INTERFACE ICylinder EXTENDS __System.IQueryInterface

PROPERTY AtHome : bool
GET
END_GET
END_PROPERTY

PROPERTY AtWork : bool
GET
END_GET
END_PROPERTY

METHOD MoveToHome : BOOL
END_METHOD

METHOD MoveToWork : BOOL
END_METHOD

PROPERTY MovingToHomePosition : BOOL
GET
END_GET
END_PROPERTY

PROPERTY MovingToWorkPosition : BOOL
GET
END_GET
END_PROPERTY

END_INTERFACE

(* stored: Version 1.1.0.1, ProductVersion 3.1.4024.4
   Itf ICylinder: Id {f5fb744e-8a3c-4ca5-afc7-036cd2bd31fb}
   Property AtHome: Id {692c9f1a-d5e3-4f4a-9a9a-282429eb8537}
   Get Get: Id {e9381276-183c-4554-9e0d-6f5dae55cf75}
   Property AtWork: Id {659097f8-ff2d-44da-ad8a-231bc9f0b243}
   Get Get: Id {835540d8-d675-47f7-a931-ab492f87d3c7}
   Method MoveToHome: Id {d6e3c3c7-b7b1-4768-b83a-9594a0e909ac}
   Method MoveToWork: Id {dd77db31-fa7d-47a7-90b5-c7891872d98e}
   Property MovingToHomePosition: Id {b6761128-8506-4c26-abb8-858156b7d17a}
   Get Get: Id {42cf0e5a-60dc-4bd6-8884-342668178fda}
   Property MovingToWorkPosition: Id {3048e18e-9228-43da-96f7-0a9368ee7049}
   Get Get: Id {f17df437-7fe7-4cb3-9c4d-2a1ed457fda4} *)
